(* CoDeSys 2.3.9.50 project: 9B.pr6 *)
(* Libraries: STANDARD.LB6 5.6.98 12:03:02 *)

(* POU MAIN, LD *)
PROGRAM MAIN
VAR
	Start AT %IX0.0: BOOL;
	ProcessON AT %QX0.0: BOOL;
	Valve_1_ON AT %QX0.1: BOOL;
	Check_Water_Level AT %IX0.1: BOOL;
	current: INT := 90;
	A AT %QX0.2: BOOL;
	Valve_2_ON AT %QX0.3: BOOL;
	B AT %QX0.4: BOOL;
	Mixer_ON AT %QX0.5: BOOL;
	T1: TON;
	Heater_ON AT %QX0.6: BOOL;
	current_temp: INT := 0;
	C AT %QX0.7: BOOL;
	Valve_3_ON AT %QX1.0: BOOL;
	D AT %QX1.1: BOOL;
END_VAR
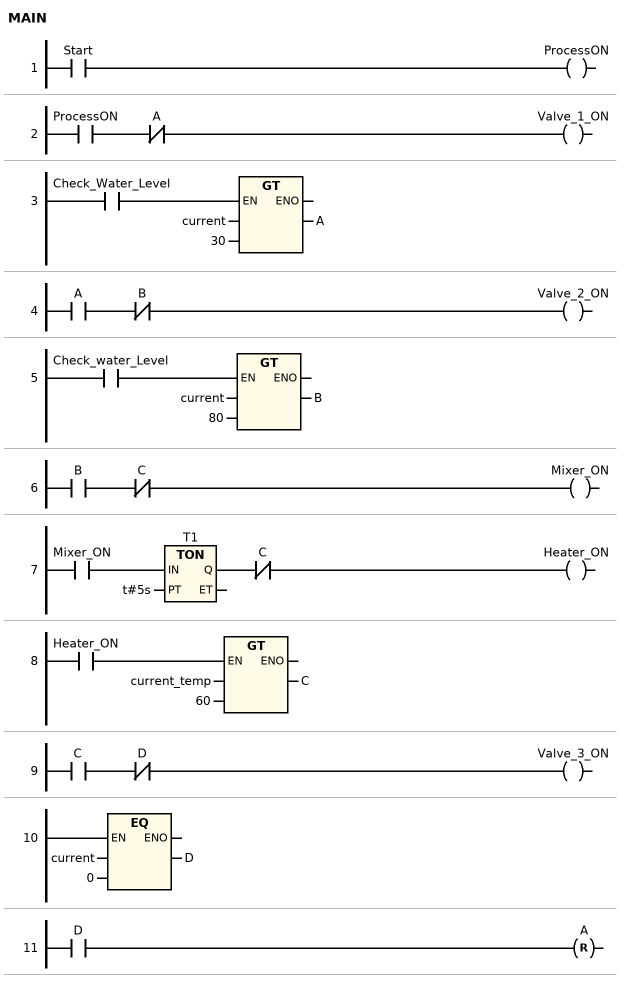
_LD_ (* Ladder Diagram *)
NETWORK 1
	[Start] --- (ProcessON)
NETWORK 2
	[ProcessON] - [/A] --- (Valve_1_ON)
NETWORK 3
	[Check_Water_Level]
		EN --- GT(current, 30) => A
NETWORK 4
	[A] - [/B] --- (Valve_2_ON)
NETWORK 5
	[Check_water_Level]
		EN --- GT(current, 80) => B
NETWORK 6
	[B] - [/C] --- (Mixer_ON)
NETWORK 7
	[Mixer_ON] - T1:TON(IN: *, PT: t#5s) - [/C] --- (Heater_ON)
NETWORK 8
	[Heater_ON]
		EN --- GT(current_temp, 60) => C
NETWORK 9
	[C] - [/D] --- (Valve_3_ON)
NETWORK 10
	*
		EN --- EQ(current, 0) => D
NETWORK 11
	[D] --- (R A)
_END_LD_
(* the same logic as Structured Text *)
(* Network 1 *)
ProcessON := Start;
(* Network 2 *)
Valve_1_ON := ProcessON AND NOT A;
(* Network 3 *)
IF Check_Water_Level THEN
	A := current > 30;
END_IF;
(* Network 4 *)
Valve_2_ON := A AND NOT B;
(* Network 5 *)
IF Check_water_Level THEN
	B := current > 80;
END_IF;
(* Network 6 *)
Mixer_ON := B AND NOT C;
(* Network 7 *)
T1(IN := Mixer_ON, PT := t#5s);
Heater_ON := T1.Q AND NOT C;
(* Network 8 *)
IF Heater_ON THEN
	C := current_temp > 60;
END_IF;
(* Network 9 *)
Valve_3_ON := C AND NOT D;
(* Network 10 *)
D := current = 0;
(* Network 11 *)
IF D THEN A := FALSE; END_IF;
END_PROGRAM
